(* Logix 5000 project; controller Traffict_Light_Limits_Instruction Emulate 5570 rev 30.12; software revision 30.01 *)

TASK T00_MainTask (continuous, watchdog 500 ms) : P00_MainProgram

MODULES
   Local : Emulate 5570 (ICP 2, rev 30.12)
      remote_controller : Emulate 5570 (ICP 4, rev 30.1, $d570ae92$ RPI 20 ms)
      Local_Communication_Card : 1756-EN2T (ICP 5, Ethernet 192.168.1.20, rev 11.1)
         Remote_Communication_Card : 1756-EN2T (Ethernet 192.168.1.21, rev 11.1, Output RPI 10 ms)
            Remote_PLC_Mill : vendor 1 type 14 code 92 (ICP 1, rev 30.1)
         Remote_Communication_Card_Assembly : 1756-EN2T (Ethernet 192.168.1.22, rev 11.1, Output RPI 10 ms)
            Digital_Remote_Input : 1756-IB16 (ICP 1, rev 3.1)
            Remote_PLC_Assembly : 1756-L72 (ICP 2, rev 30.1)
      communication_Card_Plant : 1756-EN2T (ICP 6, Ethernet 192.168.1.18, rev 11.1)
      Virtual_Module : vendor 1 type 0 code 15 (ICP 3, rev 1.1, Output RPI 50 ms)
           Local:3:C   // Phisical Memory
           Local:3:I   // Phisical Memory
           Local:3:O.Data[0].0   // Green Light
           Local:3:O.Data[0].1   // Yellow Light
           Local:3:O.Data[0].2   // Red Light
           Local:3:O   // Phisical Memory
END_MODULES

VAR_GLOBAL   (* controller tags *)
   Math_Operations : DINT[20] := ([0] := 70, [1] := 50, [2] := 1000, [3] := 2, [4] := -25, [5] := 5, [6] := 713);
   Messsages : MESSAGE;
        MessageParameters(ServiceCode := 16#004c, LocalElement := MSG_Data_Read, ...)
   Motor : BOOL;   // Virtual Memory
   MSG_Data_Read : DINT;
   Safety_SSV : BOOL;
   Start : BOOL;   // Virtual Memory
   Stop : BOOL;   // Virtual Memory
   Tag_consumed : DINT;
   WallClockTime : DINT[7] := ([0] := 2024, [1] := 2, [2] := 11, [3] := 16, [4] := 36, [5] := 1, [6] := 701276);
   WallClockTime_SSV : DINT[7];
END_VAR

PROGRAM P00_MainProgram   (* main routine R00_MainRoutine *)
VAR
   e_stop : BOOL;
   Green_Light : BOOL;
   HMI_Activated_Green_Light : BOOL;
   HMI_Activated_Red_Light : BOOL;
   HMI_Activated_Yellow_Light : BOOL;
   Manual_Automatic : BOOL;   // 1= Manual 0 = Automatic
   Red_Light : BOOL;
   safety_switch : BOOL;
   Timer : TIMER[25] := ([0].PRE := 13000);   // Control total time in each light
   Yellow_Light : BOOL;
END_VAR

ROUTINE R00_MainRoutine   (* ladder *)
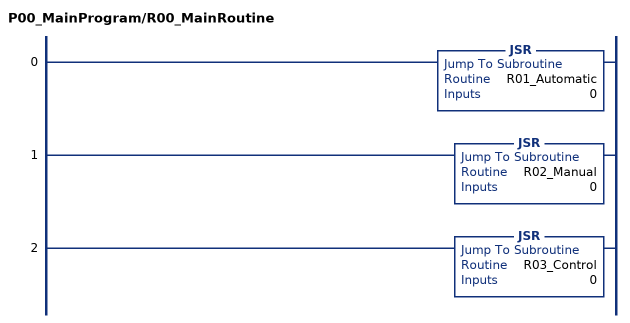
   0: JSR(R01_Automatic,0);
   1: JSR(R02_Manual,0);
   2: JSR(R03_Control,0);
END_ROUTINE

ROUTINE R01_Automatic   (* ladder *)
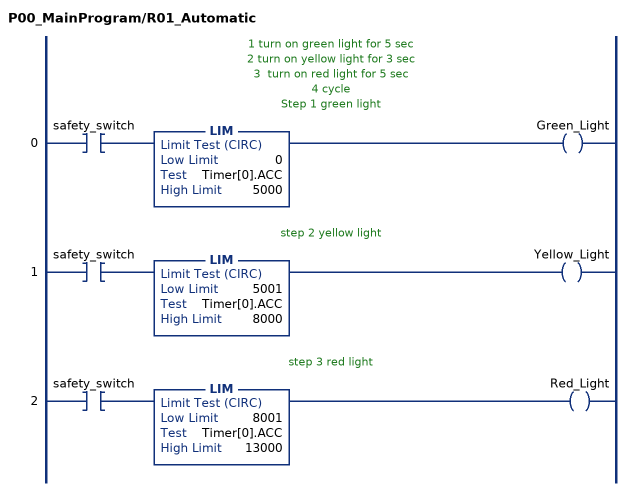
   // 1 turn on green light for 5 sec
   // 2 turn on yellow light for 3 sec
   // 3  turn on red light for 5 sec
   // 4 cycle
   // Step 1 green light
   0: XIC(safety_switch)LIM(0,Timer[0].ACC,5000)OTE(Green_Light);
   // step 2 yellow light
   1: XIC(safety_switch)LIM(5001,Timer[0].ACC,8000)OTE(Yellow_Light);
   // step 3 red light
   2: XIC(safety_switch)LIM(8001,Timer[0].ACC,13000)OTE(Red_Light);
END_ROUTINE

ROUTINE R02_Manual   (* ladder *)
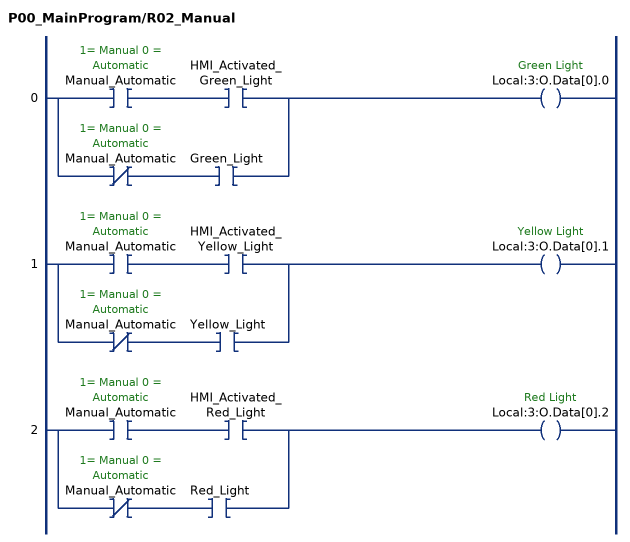
   0: [XIC(Manual_Automatic) XIC(HMI_Activated_Green_Light) ,XIO(Manual_Automatic) XIC(Green_Light) ]OTE(Local:3:O.Data[0].0);
   1: [XIC(Manual_Automatic) XIC(HMI_Activated_Yellow_Light) ,XIO(Manual_Automatic) XIC(Yellow_Light) ]OTE(Local:3:O.Data[0].1);
   2: [XIC(Manual_Automatic) XIC(HMI_Activated_Red_Light) ,XIO(Manual_Automatic) XIC(Red_Light) ]OTE(Local:3:O.Data[0].2);
END_ROUTINE

ROUTINE R03_Control   (* ladder *)
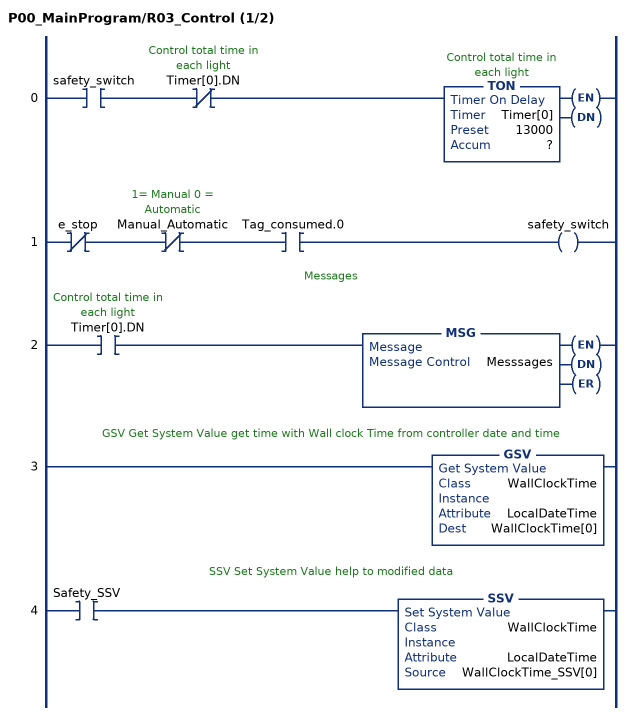
   0: XIC(safety_switch)XIO(Timer[0].DN)TON(Timer[0],?,?);
   1: XIO(e_stop)XIO(Manual_Automatic)XIC(Tag_consumed.0)OTE(safety_switch);
   // Messages
   2: XIC(Timer[0].DN)MSG(Messsages);
   // GSV Get System Value get time with Wall clock Time from controller date and time
   3: GSV(WallClockTime,,LocalDateTime,WallClockTime[0]);
   // SSV Set System Value help to modified data
   4: XIC(Safety_SSV)SSV(WallClockTime,,LocalDateTime,WallClockTime_SSV[0]);
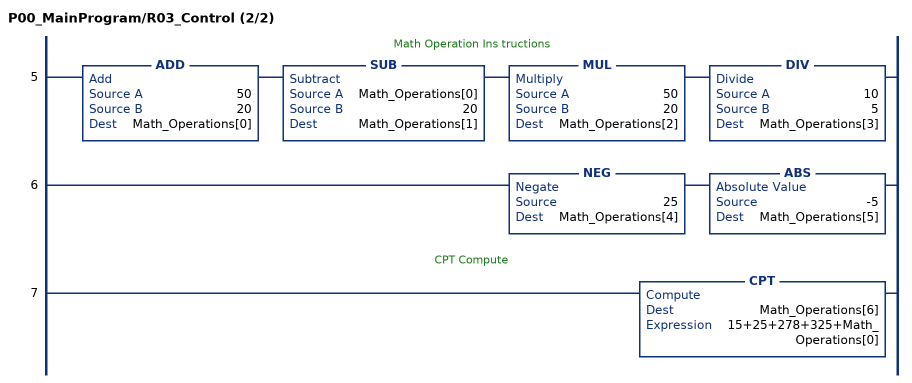
   // Math Operation Ins tructions
   5: ADD(50,20,Math_Operations[0])SUB(Math_Operations[0],20,Math_Operations[1])MUL(50,20,Math_Operations[2])DIV(10,5,Math_Operations[3]);
   6: NEG(25,Math_Operations[4])ABS(-5,Math_Operations[5]);
   // CPT Compute
   7: CPT(Math_Operations[6],15+25+278+325+Math_Operations[0]);
END_ROUTINE
END_PROGRAM
